TYPE ST_BaseHMIGroupElement_Command :
STRUCT
END_STRUCT
END_TYPE

(* stored: Version 1.1.0.1
   DUT ST_BaseHMIGroupElement_Command: Id {25789494-5929-053d-1d8c-7cab743e4d3c} *)
